// Mitsubishi GX Works2 project: 0716함수   PLC: Q02/Q02H

// global labels: Global1
VAR_GLOBAL
  공급_후 AT X0 : BOOL;
  공급_전 AT X1 : BOOL;
  드릴_상 AT X2 : BOOL;
  드릴_하 AT X3 : BOOL;
  송출_후 AT X4 : BOOL;
  송출_전 AT X5 : BOOL;
  공솔_전 AT Y20 : BOOL;
  공솔_후 AT Y21 : BOOL;
  드릴_전 AT Y22 : BOOL;
  PB1 AT X10 : BOOL;
  PB2 AT X11 : BOOL;
END_VAR

PROGRAM MAIN
VAR
  자기_1 : 업카;
  자기_2 : 업카;
  자기_3 : 업카;
  업카_1 : 업카;
END_VAR
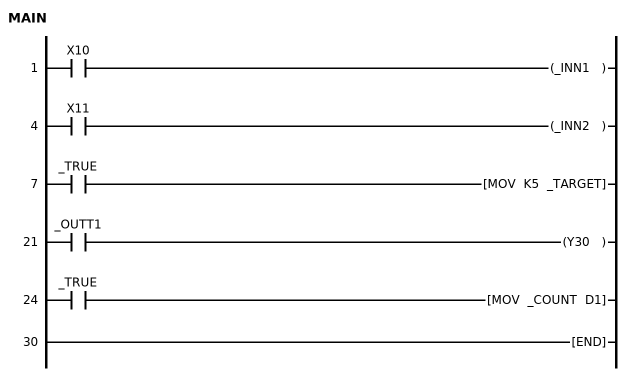
; FB BLK START 업카(업카_1)
1     LD      X10
      OUT     _INN1
4     LD      X11
      OUT     _INN2
7     LD      _TRUE
      MOV     K5 _TARGET
; FB START
; FB_NAME 업카
; INSTANCE_NAME 업카_1
; FB IN_B:INN1
; FB OUT_OUTT1:B
; FB IN_B:INN2
; FB OUT_COUNT:W
; FB IN_W:TARGET
; FB END
21    LD      _OUTT1
      OUT     Y30
24    LD      _TRUE
      MOV     _COUNT D1
; FB BLK END
30    END
END_PROGRAM

FUNCTION_BLOCK 업카
VAR_INPUT
  INN1 : BOOL;
  INN2 : BOOL;
END_VAR
VAR_OUTPUT
  OUTT1 : BOOL;
END_VAR
VAR_INPUT
  TARGET : INT;
END_VAR
VAR_OUTPUT
  COUNT : INT;
END_VAR
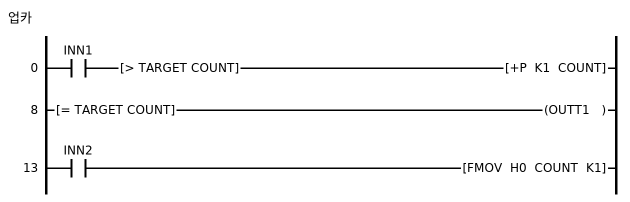
0     LD      INN1
      AND>    TARGET COUNT
      +P      K1 COUNT
8     LD=     TARGET COUNT
      OUT     OUTT1
13    LD      INN2
      FMOV    H0 COUNT K1
END_FUNCTION_BLOCK
